// TIA Portal V19 export
TYPE "SpeedMachine_Wng"
// stored: Access Published
   STRUCT
      NotAutReady : Bool;
      MissingCnd_Bkw : Bool;
      MissingCnd_Fwd : Bool;
      Ax : Struct
         Drive : Bool;
      END_STRUCT;
   END_STRUCT;
END_TYPE
